(* Logix 5000 project; controller TEC_81 vendor 1 type 14 code 148 rev 36.11; software revision 36.00; part 5 of 5 *)
(* tags used below, declared in another part *)
   Mat_1_Status : BOOL;   // General status of inputs
   Safety_Close_Loop_ok : BOOL;   // General Safety Indicator
   Safety_Mat_ok : BOOL;   // Safety Mat Close Loop Indicator
(* SafetyProgram, continued *)

ROUTINE Safety_CNC   (* ladder *)
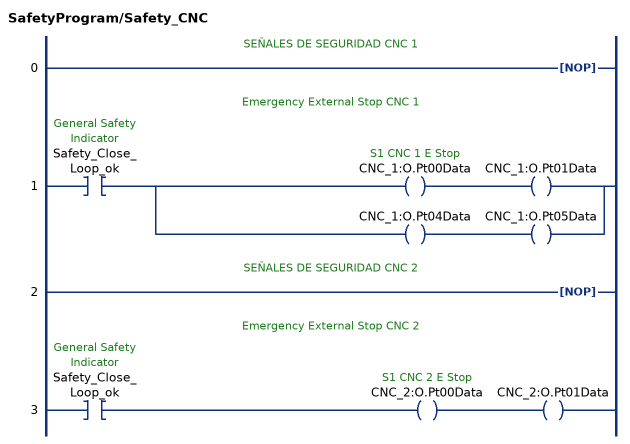
   // SEÑALES DE SEGURIDAD CNC 1
   0: NOP();
   // Emergency External Stop CNC 1
   1: XIC(Safety_Close_Loop_ok)[OTE(CNC_1:O.Pt00Data) OTE(CNC_1:O.Pt01Data) ,OTE(CNC_1:O.Pt04Data) OTE(CNC_1:O.Pt05Data) ];
   // SEÑALES DE SEGURIDAD CNC 2
   2: NOP();
   // Emergency External Stop CNC 2
   3: XIC(Safety_Close_Loop_ok)OTE(CNC_2:O.Pt00Data)OTE(CNC_2:O.Pt01Data);
END_ROUTINE

ROUTINE Safety_Mat   (* ladder *)
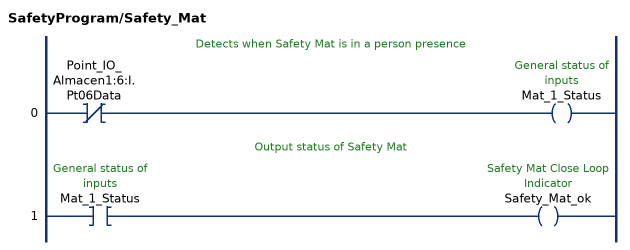
   // Detects when Safety Mat is in a person presence
   0: XIO(Point_IO_Almacen1:6:I.Pt06Data)OTE(Mat_1_Status);
   // Output status of Safety Mat
   1: XIC(Mat_1_Status)OTE(Safety_Mat_ok);
END_ROUTINE
END_PROGRAM
